// TIA Portal V21 export
VAR_GLOBAL   // PLC tag table "A0.300"
   tESTE_01 AT %I15.0 : Bool;
END_VAR
